// TIA Portal V19 export
TYPE "TetraPakV70_10_UDTNest"
   STRUCT
      OP : "OP_Int";
      Commands : "IF_Commands";
      "IF" : "TetraPakV70_10_Params";
   END_STRUCT;
END_TYPE
